FUNCTION_BLOCK FB_ModeVisualControlBox IMPLEMENTS I_ControlType
VAR_INPUT
END_VAR
VAR_OUTPUT
END_VAR
VAR
END_VAR

METHOD Joystick
VAR_INPUT
	bSwitch	: BOOL;
	bActive : BOOL;
END_VAR
IF NOT(bActive) THEN
	G_Inputs.fJoyY := 0.0;
	G_Inputs.fJoyX := 0.0;
	G_VB.fJoyX := 0.0;
	G_VB.fJoyY := 0.0;
ELSIF (bSwitch) THEN
	G_Inputs.fJoyY := G_VB.fJoyY;
	G_Inputs.fJoyX := 0.0;
	G_VB.fJoyX := 0.0;
ELSIF NOT(bSwitch) THEN
	G_Inputs.fJoyY := 0.0;
	G_Inputs.fJoyX := G_VB.fJoyX;
	G_VB.fJoyY := 0.0;
END_IF
END_METHOD

METHOD Mode
VAR_INPUT
	eCurrentMode : E_Mode;
END_VAR
G_VB.eMode := eCurrentMode;
END_METHOD

{warning 'add method implementation '}
METHOD Status
VAR_INPUT
	eStatus : E_Status;
END_VAR
G_VB.eStatus := eStatus;
END_METHOD

END_FUNCTION_BLOCK

(* stored: Version 1.1.0.1, ProductVersion 3.1.4024.12
   POU FB_ModeVisualControlBox: Id {5887b034-35fa-4339-b985-b0c482f7b634}, SpecialFunc None
   Method Joystick: Id {db07259e-d434-4bb8-906d-ae09af6d2152}
   Method Mode: Id {3fa2b439-0814-43e9-b1c7-9d95cf660055}
   Method Status: Id {15912bcb-7cba-4af3-9021-2949e1b2aceb} *)
